# B&R Automation Studio project SceneViewerCamera
Automation Studio 4.7.3.93 SP

## Configuration Config1

### Task classes (Cpu.sw)
```
Cyclic#1:
  Vis <- Vis.prg
  Trak <- Trak.prg
  SVControl <- SVControl.prg
DataObjects: McAcpSys
Binaries: FWRules, McAcpSim, arcoal, arsvcreg, TCData, McAcpDrv, arflatprv, udbdef, mvLoader, iomap, Config_1, arconfig, asfw, ashwac, sysconf, User, Role, ashwd, Config_3
Libraries: BeEasyTrak, SceneView, McBase, McAxis, McAcpTrak, standard, AsBrStr, AsMath, MpAxis, MpBase, McAcpAx, astime, powerlnk, asieccon, arssl, MpRecipe, sys_lib, runtime, FileIO
```

## Logical view

### Package Logical/Libraries - Global libraries

### Library Logical/Libraries/SceneView

#### SceneView.fun
```iecst
{REDUND_ERROR} FUNCTION_BLOCK SV_BE_MoveView (*TODO: Add your comment here*) (*$GROUP=User,$CAT=User,$GROUPICON=User.png,$CATICON=User.png*)
	VAR_INPUT
		Execute : BOOL;
		PointA : SceneViewCamera_typ;
		PointB : SceneViewCamera_typ;
		TravelTime : TIME;
	END_VAR
	VAR_OUTPUT
		Error : BOOL;
		Done : BOOL;
		SceneViewPos : SceneViewCamera_typ;
	END_VAR
	VAR
		TON_ViewChange : TON;
		State : USINT;
		ChangeRate : SceneViewCamera_typ;
	END_VAR
END_FUNCTION_BLOCK

{REDUND_ERROR} FUNCTION_BLOCK SV_BE_FocalPointMove (*TODO: Add your comment here*) (*$GROUP=User,$CAT=User,$GROUPICON=User.png,$CATICON=User.png*)
	VAR_INPUT
		FocalPointA : SceneViewCoord_typ;
		FocalPointB : SceneViewCoord_typ;
		Execute : BOOL;
		PointA : SceneViewCamera_typ;
		PointB : SceneViewCamera_typ;
		TravelTime : TIME;
		Pause : BOOL;
	END_VAR
	VAR_OUTPUT
		Error : BOOL;
		Done : BOOL;
		FocalPointPos : SceneViewCoord_typ;
		SceneViewPos : SceneViewCamera_typ;
		ElapsedTime : TIME;
		Paused : BOOL;
	END_VAR
	VAR
		TON_ViewChange : TON;
		State : USINT;
		FocalPointChangeRate : SceneViewCoord_typ;
		ChangeRate : SceneViewCamera_typ;
		RemainingTime : TIME;
		PausedTime : TIME;
	END_VAR
END_FUNCTION_BLOCK

{REDUND_ERROR} FUNCTION_BLOCK SV_BE_RadialMove
	VAR_INPUT
		FocalPointA : SceneViewCoord_typ;
		FocalPointB : SceneViewCoord_typ;
		Execute : BOOL;
		PointA : SceneViewCamera_typ;
		PointB : SceneViewCamera_typ;
		TravelTime : TIME;
		Pause : BOOL;
	END_VAR
	VAR_OUTPUT
		Error : BOOL;
		Done : BOOL;
		FocalPointPos : SceneViewCoord_typ;
		SceneViewPos : SceneViewCamera_typ;
		ElapsedTime : TIME;
	END_VAR
	VAR
		FocalPointChangeRate : SceneViewCoord_typ;
		TON_ViewChange : TON;
		State : USINT;
		ChangeRate : SceneViewCamera_typ;
		RadiusA : REAL;
		RadiusB : REAL;
		RadiusChangeRate : REAL;
		OutputRadius : REAL;
		AngleA : REAL;
		AngleB : REAL;
		AngleChangeRate : REAL;
		OutputAngle : REAL;
	END_VAR
	VAR_OUTPUT
		Paused : BOOL;
	END_VAR
	VAR
		RemainingTime : TIME;
		PausedTime : TIME;
	END_VAR
END_FUNCTION_BLOCK
```

#### SV_BE_FocalPointMove.st
```iecst
(* TODO: Add your comment here *)
FUNCTION_BLOCK SV_BE_FocalPointMove
	IF Error THEN
		State := 50;
	ELSIF NOT Execute THEN
		State := 0;
	END_IF

	CASE State OF

		0:

			ElapsedTime := T#0s;
			PausedTime := T#0s;
			Done := FALSE;
			TON_ViewChange.IN := FALSE;
		//	TON_ViewChange();

			IF Execute THEN
				IF TIME_TO_REAL(TravelTime) = 0 THEN
					Error := TRUE;
				ELSE
					SceneViewPos := PointA;
					State := 2;
				END_IF
			END_IF

		2:
			SceneViewPos.Perspective := TRUE;
			ChangeRate.Fov := (PointB.Fov - PointA.Fov) / TIME_TO_REAL(TravelTime);
			ChangeRate.Zoom := (PointB.Zoom - PointA.Zoom) / TIME_TO_REAL(TravelTime);
			ChangeRate.ViewPoint.X := (PointB.ViewPoint.X - PointA.ViewPoint.X) / TIME_TO_REAL(TravelTime);
			ChangeRate.ViewPoint.Y := (PointB.ViewPoint.Y - PointA.ViewPoint.Y) / TIME_TO_REAL(TravelTime);
			ChangeRate.ViewPoint.Z := (PointB.ViewPoint.Z - PointA.ViewPoint.Z) / TIME_TO_REAL(TravelTime);

			FocalPointChangeRate.X := (FocalPointB.X - FocalPointA.X) / TIME_TO_REAL(TravelTime);
			FocalPointChangeRate.Y := (FocalPointB.Y - FocalPointA.Y) / TIME_TO_REAL(TravelTime);
			FocalPointChangeRate.Z := (FocalPointB.Z - FocalPointA.Z) / TIME_TO_REAL(TravelTime);
			ChangeRate.OrientationVector.X := (PointB.OrientationVector.X - PointA.OrientationVector.X) / TIME_TO_REAL(TravelTime);
			ChangeRate.OrientationVector.Y := (PointB.OrientationVector.Y - PointA.OrientationVector.Y) / TIME_TO_REAL(TravelTime);
			ChangeRate.OrientationVector.Z := (PointB.OrientationVector.Z - PointA.OrientationVector.Z) / TIME_TO_REAL(TravelTime);

			TON_ViewChange.PT := TravelTime;

			State := 3;

		3:

			TON_ViewChange.IN := TRUE;

			FocalPointPos.X := (FocalPointA.X + FocalPointChangeRate.X * TIME_TO_REAL(TON_ViewChange.ET));
			FocalPointPos.Y := (FocalPointA.Y + FocalPointChangeRate.Y * TIME_TO_REAL(TON_ViewChange.ET));
			FocalPointPos.Z := (FocalPointA.Z + FocalPointChangeRate.Z * TIME_TO_REAL(TON_ViewChange.ET));

			SceneViewPos.OrientationVector.X := PointA.OrientationVector.X + ChangeRate.OrientationVector.X * TIME_TO_REAL(TON_ViewChange.ET);
			SceneViewPos.OrientationVector.Y := PointA.OrientationVector.Y + ChangeRate.OrientationVector.Y * TIME_TO_REAL(TON_ViewChange.ET);
			SceneViewPos.OrientationVector.Z := PointA.OrientationVector.Z + ChangeRate.OrientationVector.Z * TIME_TO_REAL(TON_ViewChange.ET);

			SceneViewPos.Fov := PointA.Fov + ChangeRate.Fov * TIME_TO_REAL(TON_ViewChange.ET);
			SceneViewPos.Zoom := PointA.Zoom + ChangeRate.Zoom * TIME_TO_REAL(TON_ViewChange.ET);
			SceneViewPos.ViewPoint.X := PointA.ViewPoint.X + ChangeRate.ViewPoint.X * TIME_TO_REAL(TON_ViewChange.ET);
			SceneViewPos.ViewPoint.Y := PointA.ViewPoint.Y + ChangeRate.ViewPoint.Y * TIME_TO_REAL(TON_ViewChange.ET);
			SceneViewPos.ViewPoint.Z := PointA.ViewPoint.Z + ChangeRate.ViewPoint.Z * TIME_TO_REAL(TON_ViewChange.ET);
			SceneViewPos.ViewVector.X := (FocalPointPos.X - SceneViewPos.ViewPoint.X) / 1000.0;
			SceneViewPos.ViewVector.Y := (FocalPointPos.Y - SceneViewPos.ViewPoint.Y) / 1000.0;
			SceneViewPos.ViewVector.Z := (FocalPointPos.Z - SceneViewPos.ViewPoint.Z) / 1000.0;

			ElapsedTime := TON_ViewChange.ET + PausedTime;

			IF TON_ViewChange.Q THEN
				TON_ViewChange.IN := FALSE;
				State := 4;
			ELSIF Pause THEN
				FocalPointA.X := FocalPointPos.X;
				FocalPointA.Y := FocalPointPos.Y;
				FocalPointA.Z := FocalPointPos.Z;
				PointA.OrientationVector.X := SceneViewPos.OrientationVector.X;
				PointA.OrientationVector.Y := SceneViewPos.OrientationVector.Y;
				PointA.OrientationVector.Z := SceneViewPos.OrientationVector.Z;
				PointA.Fov := SceneViewPos.Fov;
				PointA.Zoom := SceneViewPos.Zoom;
				PointA.ViewPoint.X := SceneViewPos.ViewPoint.X;
				PointA.ViewPoint.Y := SceneViewPos.ViewPoint.Y;
				PointA.ViewPoint.Z := SceneViewPos.ViewPoint.Z;

				RemainingTime := TravelTime - ElapsedTime;
				PausedTime := ElapsedTime;
				TON_ViewChange.PT := RemainingTime;

				TON_ViewChange.IN := FALSE;
				State := 10;
			END_IF

		//	TON_ViewChange();

		4:

			Done := TRUE;

		10:
			Paused := TRUE;
			IF NOT Pause THEN
				Paused := FALSE;
				Pause := FALSE;
				State := 3;
			END_IF

		50:
			IF NOT Execute THEN
				Error := FALSE;
				State := 0;
			END_IF

	END_CASE

	TON_ViewChange();

END_FUNCTION_BLOCK
```

#### SV_BE_RadialMove.st
```iecst
(* TODO: Add your comment here *)
FUNCTION_BLOCK SV_BE_RadialMove
	IF Error THEN
		State := 50;
	ELSIF NOT Execute THEN
		State := 0;
	END_IF

	CASE State OF
		0:
			ElapsedTime := T#0s;
			PausedTime := T#0s;
			Done := FALSE;
			TON_ViewChange.IN := FALSE;

			IF Execute THEN
				IF (TIME_TO_REAL(TravelTime) = 0) THEN
					Error := TRUE;
				ELSE
					SceneViewPos := PointA;
					State := 1;
				END_IF
			END_IF

		1:

			AngleA := atan2((PointA.ViewPoint.Y - FocalPointA.Y),(PointA.ViewPoint.X - FocalPointA.X));
			AngleB := atan2((PointB.ViewPoint.Y - FocalPointB.Y),(PointB.ViewPoint.X - FocalPointB.X));

			RadiusA := (PointA.ViewPoint.X - FocalPointA.X) / COS(AngleA);
			RadiusB := (PointB.ViewPoint.X - FocalPointB.X) / COS(AngleB);

			SceneViewPos.Perspective := TRUE;

			RadiusChangeRate := (RadiusB - RadiusA) / TIME_TO_REAL(TravelTime);
			AngleChangeRate := (AngleB - AngleA) / TIME_TO_REAL(TravelTime);
			ChangeRate.Fov := (PointB.Fov - PointA.Fov) / TIME_TO_REAL(TravelTime);
			ChangeRate.Zoom := (PointB.Zoom - PointA.Zoom) / TIME_TO_REAL(TravelTime);
			ChangeRate.ViewPoint.X := (PointB.ViewPoint.X - PointA.ViewPoint.X) / TIME_TO_REAL(TravelTime);
			ChangeRate.ViewPoint.Y := (PointB.ViewPoint.Y - PointA.ViewPoint.Y) / TIME_TO_REAL(TravelTime);
			ChangeRate.ViewPoint.Z := (PointB.ViewPoint.Z - PointA.ViewPoint.Z) / TIME_TO_REAL(TravelTime);
			ChangeRate.OrientationVector.X := (PointB.OrientationVector.X - PointA.OrientationVector.X) / TIME_TO_REAL(TravelTime);
			ChangeRate.OrientationVector.Y := (PointB.OrientationVector.Y - PointA.OrientationVector.Y) / TIME_TO_REAL(TravelTime);
			ChangeRate.OrientationVector.Z := (PointB.OrientationVector.Z - PointA.OrientationVector.Z) / TIME_TO_REAL(TravelTime);
			FocalPointChangeRate.X := (FocalPointB.X - FocalPointA.X) / TIME_TO_REAL(TravelTime);
			FocalPointChangeRate.Y := (FocalPointB.Y - FocalPointA.Y) / TIME_TO_REAL(TravelTime);
			FocalPointChangeRate.Z := (FocalPointB.Z - FocalPointA.Z) / TIME_TO_REAL(TravelTime);

			TON_ViewChange.PT := TravelTime;
			State := 2;

		2:

			TON_ViewChange.IN := TRUE;

			FocalPointPos.X := (FocalPointA.X + FocalPointChangeRate.X * TIME_TO_REAL(TON_ViewChange.ET));
			FocalPointPos.Y := (FocalPointA.Y + FocalPointChangeRate.Y * TIME_TO_REAL(TON_ViewChange.ET));
			FocalPointPos.Z := (FocalPointA.Z + FocalPointChangeRate.Z * TIME_TO_REAL(TON_ViewChange.ET));

			OutputAngle := AngleA + AngleChangeRate * TIME_TO_REAL(TON_ViewChange.ET);
			OutputRadius := RadiusA + RadiusChangeRate * TIME_TO_REAL(TON_ViewChange.ET);

			SceneViewPos.ViewPoint.X := (OutputRadius * COS(OutputAngle)) + FocalPointPos.X;
			SceneViewPos.ViewPoint.Y := (OutputRadius * SIN(OutputAngle)) + FocalPointPos.Y;

			SceneViewPos.Fov := PointA.Fov + ChangeRate.Fov * TIME_TO_REAL(TON_ViewChange.ET);
			SceneViewPos.Zoom := PointA.Zoom + ChangeRate.Zoom * TIME_TO_REAL(TON_ViewChange.ET);
			SceneViewPos.ViewPoint.Z := PointA.ViewPoint.Z + ChangeRate.ViewPoint.Z * TIME_TO_REAL(TON_ViewChange.ET);
			SceneViewPos.ViewVector.X := (FocalPointPos.X - SceneViewPos.ViewPoint.X) / 1000.0;
			SceneViewPos.ViewVector.Y := (FocalPointPos.Y - SceneViewPos.ViewPoint.Y) / 1000.0;
			SceneViewPos.ViewVector.Z := (FocalPointPos.Z - SceneViewPos.ViewPoint.Z) / 1000.0;
			SceneViewPos.OrientationVector.X := PointA.OrientationVector.X + ChangeRate.OrientationVector.X * TIME_TO_REAL(TON_ViewChange.ET);
			SceneViewPos.OrientationVector.Y := PointA.OrientationVector.Y + ChangeRate.OrientationVector.Y * TIME_TO_REAL(TON_ViewChange.ET);
			SceneViewPos.OrientationVector.Z := PointA.OrientationVector.Z + ChangeRate.OrientationVector.Z * TIME_TO_REAL(TON_ViewChange.ET);

			ElapsedTime := TON_ViewChange.ET + PausedTime;

			IF TON_ViewChange.Q THEN
				TON_ViewChange.IN := FALSE;
				State := 3;
			ELSIF Pause THEN
				FocalPointA.X := FocalPointPos.X;
				FocalPointA.Y := FocalPointPos.Y;
				FocalPointA.Z := FocalPointPos.Z;
				AngleA := OutputAngle;
				RadiusA := OutputRadius;

				PointA.OrientationVector.X := SceneViewPos.OrientationVector.X;
				PointA.OrientationVector.Y := SceneViewPos.OrientationVector.Y;
				PointA.OrientationVector.Z := SceneViewPos.OrientationVector.Z;
				PointA.Fov := SceneViewPos.Fov;
				PointA.Zoom := SceneViewPos.Zoom;
				PointA.ViewPoint.Z := SceneViewPos.ViewPoint.Z;

				RemainingTime := TravelTime - ElapsedTime;
				PausedTime := ElapsedTime;
				TON_ViewChange.PT := RemainingTime;

				TON_ViewChange.IN := FALSE;
				State := 10;
			END_IF

		3:
			Done := TRUE;

		10:
			Paused := TRUE;
			IF NOT Pause THEN
				Paused := FALSE;
				Pause := FALSE;
				State := 2;
			END_IF

		50:
			IF NOT Execute THEN
				Error := FALSE;
				State := 0;
			END_IF

	END_CASE

	TON_ViewChange();

END_FUNCTION_BLOCK
```

### Program Logical/SVControl (IEC)

#### Types.typ
```iecst
TYPE
	MoveType_enum :
		(
		LINEAR,
		RADIAL
		);
	Binding_typ : 	STRUCT
		Camera : SceneViewCamera_typ;
		FocalPoint : SceneViewCoord_typ;
		FocalPointVisible : BOOL;
	END_STRUCT;
	Vis_typ : 	STRUCT
		Controls : Controls_typ;
		Bind : Binding_typ;
	END_STRUCT;
	LinearControls_typ : 	STRUCT
		XBtnPos : USINT;
		XBtnNeg : USINT;
		YBtnPos : USINT;
		YBtnNeg : USINT;
		Y : REAL;
		X : REAL;
	END_STRUCT;
	CircularControls_typ : 	STRUCT
		RadiusBtnNeg : USINT;
		RadiusBtnPos : USINT;
		Angle : REAL;
		Radius : REAL;
	END_STRUCT;
	Controls_typ : 	STRUCT
		FocalPoint : FocalPointControls_typ;
		Fov : REAL;
		Z : REAL;
		Circular : CircularControls_typ;
		Linear : LinearControls_typ;
		SavePointA : BOOL;
		MoveType : USINT;
		NewMove : BOOL;
		Start : BOOL;
		Load : BOOL;
		Save : BOOL;
		SelectedMove : USINT;
		MoveMode : MoveType_enum;
		TimeInput : REAL;
		ActiveMoveTravelTime : TIME;
		ActiveMoveElapsedTime : TIME;
		Pause : BOOL;
		Stop : BOOL;
	END_STRUCT;
	FocalPointControls_typ : 	STRUCT
		XBtnPos : USINT;
		XBtnNeg : USINT;
		YBtnPos : USINT;
		YBtnNeg : USINT;
		ZBtnPos : USINT;
		ZBtnNeg : USINT;
		Visible : BOOL;
	END_STRUCT;
	Move_typ : 	STRUCT
		IsSaved : BOOL;
		MoveType : MoveType_enum;
		Point : SceneViewCamera_typ;
		FocalPoint : SceneViewCoord_typ;
		TravelTime : TIME;
	END_STRUCT;
	State_enum :
		(
		MOVE_SETTINGS,
		NEW_MOVE,
		UPDATE_LIST,
		REBUILD_LIST,
		NEW_MOVE_SAVE,
		SAVE_MOVE,
		LOAD_MOVE,
		START_MOVE,
		LINEAR_MOVE,
		WAIT_FOR_LINEAR_MOVE_DONE,
		RADIAL_MOVE,
		WAIT_FOR_RADIAL_MOVE_DONE,
		MOVE_COMPLETE,
		SAVE_LOAD_RECIPE,
		WAIT_FOR_STOP
		);
	RecipeCtrlTyp : 	STRUCT
		Cmd : RecipeCtrlCmdTyp;
		Par : RecipeCtrlParTyp;
		Sts : RecipeCtrlStsTyp;
	END_STRUCT;
	RecipeCtrlCmdTyp : 	STRUCT
		Save : BOOL;
		Load : BOOL;
	END_STRUCT;
	RecipeCtrlParTyp : 	STRUCT
		FileName : STRING[80];
	END_STRUCT;
	RecipeCtrlStsTyp : 	STRUCT
		LastLoadedRecipe : STRING[80];
	END_STRUCT;
END_TYPE
```

#### Main.st
```iecst
PROGRAM _INIT
	(* Insert code here *)

	Point[0] := StartView;
	Vis.Bind.Camera := StartView;

	Vis.Bind.FocalPoint.X := FocalPointInit.X;
	Vis.Bind.FocalPoint.Y := FocalPointInit.Y;
	Vis.Bind.FocalPoint.Z := FocalPointInit.Z;

	Vis.Controls.Linear.X := StartView.ViewPoint.X;
	Vis.Controls.Linear.Y := StartView.ViewPoint.Y;
	Vis.Controls.Z := StartView.ViewPoint.Z;
	Vis.Controls.Fov := StartView.Fov;
	Vis.Controls.Circular.Radius := 100;

	SvMovieRecipeFb.MpLink := ADR(gRecipeScnViewer);
	SvMovieRecipeFb.Enable := TRUE;
	SvMovieRecipeFb.Category := ADR('SvMovie');
	SvMovieRecipeFb.DeviceName := ADR('SvMovie');
	SvMovieRecipeFb.FileName := ADR(svMovieRecipeIf.Par.FileName);
	SvMovieRecipeFb();

	SvMovieRecipeRegParFb.MpLink := ADR(gRecipeScnViewer);
	SvMovieRecipeRegParFb.Enable := TRUE;
	SvMovieRecipeRegParFb.Category := ADR('SvMovie');
	SvMovieRecipeRegParFb.PVName := ADR('SVControl:CamMove');
	SvMovieRecipeRegParFb();
END_PROGRAM

PROGRAM _CYCLIC
	Vis.Bind.FocalPoint.X := Vis.Bind.FocalPoint.X + Vis.Controls.FocalPoint.XBtnPos - Vis.Controls.FocalPoint.XBtnNeg;
	Vis.Bind.FocalPoint.Y := Vis.Bind.FocalPoint.Y + Vis.Controls.FocalPoint.YBtnPos - Vis.Controls.FocalPoint.YBtnNeg;
	Vis.Bind.FocalPoint.Z := Vis.Bind.FocalPoint.Z + Vis.Controls.FocalPoint.ZBtnPos - Vis.Controls.FocalPoint.ZBtnNeg;

	Vis.Controls.Circular.Radius := Vis.Controls.Circular.Radius + Vis.Controls.Circular.RadiusBtnPos - Vis.Controls.Circular.RadiusBtnNeg;
	Vis.Controls.Linear.X := Vis.Controls.Linear.X + Vis.Controls.Linear.XBtnPos - Vis.Controls.Linear.XBtnNeg;
	Vis.Controls.Linear.Y := Vis.Controls.Linear.Y + Vis.Controls.Linear.YBtnPos - Vis.Controls.Linear.YBtnNeg;

	Vis.Bind.FocalPointVisible := Vis.Controls.FocalPoint.Visible;

	CASE State OF
		MOVE_SETTINGS: //set points
			CASE Vis.Controls.MoveMode OF
				LINEAR:
					MoveText := 'Linear';
					Vis.Bind.Camera.ViewPoint.X := Vis.Controls.Linear.X;
					Vis.Bind.Camera.ViewPoint.Y := Vis.Controls.Linear.Y;

					//keeps view the same when switching to radial mode
					AngleRad := atan2((Vis.Bind.Camera.ViewPoint.Y - Vis.Bind.FocalPoint.Y),(Vis.Bind.Camera.ViewPoint.X - Vis.Bind.FocalPoint.X));
					Vis.Controls.Circular.Angle := AngleRad * 180 / PI;
					IF Vis.Controls.Circular.Angle < 0 THEN
						Vis.Controls.Circular.Angle := Vis.Controls.Circular.Angle + 360;
					ELSIF Vis.Controls.Circular.Angle >= 360 THEN
						Vis.Controls.Circular.Angle := Vis.Controls.Circular.Angle - 360;
					END_IF
					Vis.Controls.Circular.Radius := (Vis.Bind.Camera.ViewPoint.X - Vis.Bind.FocalPoint.X) / COS(AngleRad);
				RADIAL:
					MoveText := 'Radial';
					AngleRad := Vis.Controls.Circular.Angle * PI / 180;

					Vis.Bind.Camera.ViewPoint.X := (Vis.Controls.Circular.Radius * COS(AngleRad)) + Vis.Bind.FocalPoint.X;
					Vis.Bind.Camera.ViewPoint.Y := (Vis.Controls.Circular.Radius * SIN(AngleRad)) + Vis.Bind.FocalPoint.Y;

					Vis.Controls.Linear.X := Vis.Bind.Camera.ViewPoint.X;
					Vis.Controls.Linear.Y := Vis.Bind.Camera.ViewPoint.Y;
			END_CASE

			Vis.Bind.Camera.OrientationVector.X := 0;
			Vis.Bind.Camera.OrientationVector.Y := 0;
			Vis.Bind.Camera.OrientationVector.Z := 1;

			Vis.Bind.Camera.ViewPoint.Z := Vis.Controls.Z;
			Vis.Bind.Camera.Fov := Vis.Controls.Fov;

			Vis.Bind.Camera.ViewVector.X := (Vis.Bind.FocalPoint.X - Vis.Bind.Camera.ViewPoint.X) / 1000.0;
			Vis.Bind.Camera.ViewVector.Y := (Vis.Bind.FocalPoint.Y - Vis.Bind.Camera.ViewPoint.Y) / 1000.0;
			Vis.Bind.Camera.ViewVector.Z := (Vis.Bind.FocalPoint.Z - Vis.Bind.Camera.ViewPoint.Z) / 1000.0;

			IF Vis.Controls.NewMove THEN
				Vis.Controls.NewMove := FALSE;
				State := NEW_MOVE;
			ELSIF Vis.Controls.Load THEN
				State := LOAD_MOVE;
			ELSIF Vis.Controls.Save THEN
				Vis.Controls.Save := FALSE;
				State := SAVE_MOVE;
			END_IF

			IF svMovieRecipeIf.Cmd.Load OR svMovieRecipeIf.Cmd.Save THEN
				SvMovieRecipeFb.Save := svMovieRecipeIf.Cmd.Save;
				SvMovieRecipeFb.Load := svMovieRecipeIf.Cmd.Load;

				State := SAVE_LOAD_RECIPE;
			END_IF

			IF Vis.Controls.SavePointA THEN
				Vis.Controls.SavePointA := FALSE;
				Point[0] := Vis.Bind.Camera;
			END_IF

			IF Vis.Controls.Start  THEN
				IF (TotalNumMoves > 0) THEN
					CompletedMoves := 0;
					PointA := Point[0];
					PointB := CamMove[0].Point;
					FocalPointA := FocalPointInit;
					FocalPointB := CamMove[0].FocalPoint;
					State := START_MOVE;
				ELSE
					Vis.Controls.Start := FALSE;
				END_IF
			END_IF

		NEW_MOVE: //new move
			FOR i := 0 TO MAX_NUM_MOVES DO
				IF NOT CamMove[i].IsSaved THEN
					CamMove[i].IsSaved := TRUE;
					CamMove[i].MoveType := Vis.Controls.MoveMode;
					CamMove[i].TravelTime := REAL_TO_TIME(Vis.Controls.TimeInput * 1000);

					State := NEW_MOVE_SAVE;
					EXIT;
				ELSIF i = MAX_NUM_MOVES THEN
					State := MOVE_SETTINGS;
				END_IF
			END_FOR

		NEW_MOVE_SAVE:

			TotalNumMoves := TotalNumMoves + 1;
			CamMove[i].Point := Vis.Bind.Camera;
			CamMove[i].FocalPoint := Vis.Bind.FocalPoint;

			State := UPDATE_LIST;

		UPDATE_LIST:
			brsftoa(i, ADR(MoveIndexString));
			MoveNumText[i] := CONCAT(MoveIndexString, ': ');
			MoveNumText[i] := CONCAT(MoveNumText[i], MoveText);
			MoveNumText[i] := CONCAT(MoveNumText[i], ' Move');

			IntermediateDateProvider[i] := CONCAT('{"value":"',MoveIndexString);
			IntermediateDateProvider[i] := CONCAT(IntermediateDateProvider[i],'","text":"');
			IntermediateDateProvider[i] := CONCAT(IntermediateDateProvider[i], MoveNumText[i]);
			DataProvider[i] := CONCAT(IntermediateDateProvider[i],'"}');

			State := MOVE_SETTINGS;
		SAVE_LOAD_RECIPE:
			IF SvMovieRecipeFb.CommandDone THEN
				IF svMovieRecipeIf.Cmd.Load THEN
					SvMovieRecipeFb.Load := FALSE;
					svMovieRecipeIf.Cmd.Load := FALSE;
					svMovieRecipeIf.Sts.LastLoadedRecipe := svMovieRecipeIf.Par.FileName;

					State := REBUILD_LIST;
				ELSIF svMovieRecipeIf.Cmd.Save THEN
					SvMovieRecipeFb.Save := FALSE;
					svMovieRecipeIf.Cmd.Save := FALSE;

					State := MOVE_SETTINGS;
				END_IF
			END_IF
		REBUILD_LIST:
			brsmemset(ADR(DataProvider),0,SIZEOF(DataProvider));
			brsmemset(ADR(MoveNumText),0,SIZEOF(MoveNumText));
			brsmemset(ADR(IntermediateDateProvider),0,SIZEOF(IntermediateDateProvider));
			TotalNumMoves := 0; //Added for loading saved recipes
			FOR i:=0 TO MAX_NUM_MOVES DO
				IF CamMove[i].IsSaved THEN
					TotalNumMoves := TotalNumMoves + 1;
					brsftoa(i, ADR(MoveIndexString));
					MoveNumText[i] := CONCAT(MoveIndexString, ': ');
					CASE CamMove[i].MoveType OF
						LINEAR:
							MoveNumText[i] := CONCAT(MoveNumText[i], 'Linear');
						RADIAL:
							MoveNumText[i] := CONCAT(MoveNumText[i], 'Radial');
					END_CASE;
					MoveNumText[i] := CONCAT(MoveNumText[i], ' Move');

					IntermediateDateProvider[i] := CONCAT('{"value":"',MoveIndexString);
					IntermediateDateProvider[i] := CONCAT(IntermediateDateProvider[i],'","text":"');
					IntermediateDateProvider[i] := CONCAT(IntermediateDateProvider[i], MoveNumText[i]);
					DataProvider[i] := CONCAT(IntermediateDateProvider[i],'"}');
				END_IF
			END_FOR;

			State := MOVE_SETTINGS;
		LOAD_MOVE: //load
			Vis.Controls.Load := FALSE;

			IF CamMove[Vis.Controls.SelectedMove].IsSaved THEN
				Vis.Controls.Linear.X := CamMove[Vis.Controls.SelectedMove].Point.ViewPoint.X;
				Vis.Controls.Linear.Y := CamMove[Vis.Controls.SelectedMove].Point.ViewPoint.Y;

				Vis.Controls.Z := CamMove[Vis.Controls.SelectedMove].Point.ViewPoint.Z;
				Vis.Controls.Fov := CamMove[Vis.Controls.SelectedMove].Point.Fov;
				Vis.Controls.TimeInput := TIME_TO_REAL(CamMove[Vis.Controls.SelectedMove].TravelTime) / 1000;
				Vis.Controls.MoveMode := CamMove[Vis.Controls.SelectedMove].MoveType;

				Vis.Bind.Camera := CamMove[Vis.Controls.SelectedMove].Point;
				Vis.Bind.FocalPoint := CamMove[Vis.Controls.SelectedMove].FocalPoint;

				//update radial controls
				AngleRad := atan2((Vis.Bind.Camera.ViewPoint.Y - Vis.Bind.FocalPoint.Y),(Vis.Bind.Camera.ViewPoint.X - Vis.Bind.FocalPoint.X));
				Vis.Controls.Circular.Angle := AngleRad * 180 / PI;
				IF Vis.Controls.Circular.Angle < 0 THEN
					Vis.Controls.Circular.Angle := Vis.Controls.Circular.Angle + 360;
				ELSIF Vis.Controls.Circular.Angle >= 360 THEN
					Vis.Controls.Circular.Angle := Vis.Controls.Circular.Angle - 360;
				END_IF
				Vis.Controls.Circular.Radius := (Vis.Bind.Camera.ViewPoint.X - Vis.Bind.FocalPoint.X) / COS(AngleRad);

			END_IF
			State := MOVE_SETTINGS;

		SAVE_MOVE: //save
			IF CamMove[Vis.Controls.SelectedMove].IsSaved THEN
				CamMove[Vis.Controls.SelectedMove].Point := Vis.Bind.Camera;
				CamMove[Vis.Controls.SelectedMove].FocalPoint := Vis.Bind.FocalPoint;
				CamMove[Vis.Controls.SelectedMove].TravelTime := REAL_TO_TIME(Vis.Controls.TimeInput * 1000);
				i := Vis.Controls.SelectedMove;
				State := UPDATE_LIST;
			ELSE
				State := MOVE_SETTINGS;
			END_IF

		START_MOVE:
			TravelTime := CamMove[CompletedMoves].TravelTime;
			IF CamMove[CompletedMoves].MoveType = LINEAR THEN
				State := LINEAR_MOVE;
			ELSIF CamMove[CompletedMoves].MoveType = RADIAL THEN
				State := RADIAL_MOVE;
			END_IF

		RADIAL_MOVE:
			Vis.Controls.SelectedMove := CompletedMoves;
			RadialMove.PointA := PointA;
			RadialMove.PointB := PointB;
			RadialMove.FocalPointA := FocalPointA;
			RadialMove.FocalPointB := FocalPointB;
			RadialMove.TravelTime := TravelTime;
			RadialMove.Execute := TRUE;
			State := WAIT_FOR_RADIAL_MOVE_DONE;

		WAIT_FOR_RADIAL_MOVE_DONE:

			RadialMove.Pause := Vis.Controls.Pause;

			Vis.Controls.ActiveMoveTravelTime := TravelTime;
			Vis.Controls.ActiveMoveElapsedTime := RadialMove.ElapsedTime;
			Vis.Bind.FocalPoint := RadialMove.FocalPointPos;
			Vis.Bind.Camera := RadialMove.SceneViewPos;

			IF RadialMove.Done THEN
				RadialMove.Execute := FALSE;
				CompletedMoves := CompletedMoves + 1;
				State := MOVE_COMPLETE;
			ELSIF Vis.Controls.Stop THEN
				Vis.Controls.Stop := FALSE;
				RadialMove.Execute := FALSE;
				CompletedMoves := TotalNumMoves;
				State := MOVE_COMPLETE;
			END_IF

		LINEAR_MOVE:
			Vis.Controls.SelectedMove := CompletedMoves;
			FocalPointMove.PointA := PointA;
			FocalPointMove.PointB := PointB;
			FocalPointMove.FocalPointA := FocalPointA;
			FocalPointMove.FocalPointB := FocalPointB;
			FocalPointMove.TravelTime := TravelTime;
			FocalPointMove.Execute := TRUE;
			State := WAIT_FOR_LINEAR_MOVE_DONE;

		WAIT_FOR_LINEAR_MOVE_DONE:

			FocalPointMove.Pause := Vis.Controls.Pause;

			Vis.Controls.ActiveMoveTravelTime := TravelTime;
			Vis.Controls.ActiveMoveElapsedTime := FocalPointMove.ElapsedTime;
			Vis.Bind.FocalPoint := FocalPointMove.FocalPointPos;
			Vis.Bind.Camera := FocalPointMove.SceneViewPos;

			IF FocalPointMove.Done THEN
				FocalPointMove.Execute := FALSE;
				CompletedMoves := CompletedMoves + 1;
				State := MOVE_COMPLETE;
			ELSIF Vis.Controls.Stop THEN
				Vis.Controls.Stop := FALSE;
				FocalPointMove.Execute := FALSE;
				CompletedMoves := TotalNumMoves;
				State := MOVE_COMPLETE;
			END_IF

		MOVE_COMPLETE:
			IF CompletedMoves < TotalNumMoves THEN
				PointA := Vis.Bind.Camera;
				PointB := CamMove[CompletedMoves].Point;
				FocalPointA := Vis.Bind.FocalPoint;
				FocalPointB := CamMove[CompletedMoves].FocalPoint;
				State := START_MOVE;
			ELSE
				Vis.Controls.ActiveMoveElapsedTime := T#0s;
				Vis.Controls.Start := FALSE;
				Vis.Controls.Pause := FALSE;
				State := MOVE_SETTINGS;
			END_IF

	END_CASE

	FocalPointMove();
	RadialMove();
	SvMovieRecipeFb();
	SvMovieRecipeRegParFb();

END_PROGRAM

PROGRAM _EXIT
	(* Insert code here *)

END_PROGRAM
```

- Visualisation Logical/mappView (not shown)

Listed in the project but not available here: Logical/Global.typ, Logical/Segments.var, Logical/Global.var, Logical/Vis, Logical/Trak, Logical/SavedMovies
